Staubli VAL3: PLC.dtx

public num nToSuperV
string sProgList
string sPresetList
string listProgram
public jointRx jHome
public mdesc nom_speed = {rmax=9999, blend=off}
string sSessionList
string sPalletName
string sSession
string sSession2
dio dOutRobIsReady = {link=ApplicomIO-1\TOPIC1_A-BLOCKA\%Q1}
dio dOutRobInHome = {link=ApplicomIO-1\TOPIC1_A-BLOCKA\%Q0}
dio dOutRobCycle = {link=ApplicomIO-1\TOPIC1_A-BLOCKA\%Q2}
dio dOutRobErr = {link=ApplicomIO-1\TOPIC1_A-BLOCKA\%Q4}
dio dInCycle = {link=ApplicomIO-1\TOPIC1_A-BLOCKA\%I0}
bool bError
aio aSelect = {link=ApplicomIO-1\TOPIC1_A-BLOCKA\%IW8}
num nProgCode
string sProgName
dio dInPlcErr = {link=ApplicomIO-1\TOPIC1_A-BLOCKA\%I1}
dio dOutGunOn = {link=valve1}
dio dOutJobDone
dio dInGohome = {link=ApplicomIO-1\TOPIC1_A-BLOCKA\%I4}
dio dInPauseCycle = {link=ApplicomIO-1\TOPIC1_A-BLOCKA\%I2}
dio dInResumeCycle = {link=ApplicomIO-1\TOPIC1_A-BLOCKA\%I3}
dio dIndisablepower = {link=ApplicomIO-1\TOPIC1_A-BLOCKA\%I5}
dio dOutPauseCycle = {link=ApplicomIO-1\TOPIC1_A-BLOCKA\%Q3}
public aio aTime = {link=ApplicomIO-1\TOPIC1_A-BLOCKA\%QW8}
public aio aSudu = {link=ApplicomIO-1\TOPIC1_A-BLOCKA\%IW10}
